{attribute 'enable_dynamic_creation'}
FUNCTION_BLOCK FB_AxisMoveCommand IMPLEMENTS I_Command
VAR
	_Axis : I_Axis;
	_Target : REAL;
	_Description : STRING;
END_VAR

{attribute 'monitoring' := 'call'}
PROPERTY Description : STRING
GET
Description := _Description;
END_GET
END_PROPERTY

METHOD Execute : E_Progress
_Axis.MoveAbsolute(_target);

Execute := E_Progress.Completed;
END_METHOD

//FB_Init is always available implicitly and it is used primarily for initialization.
//The return value is not evaluated. For a specific influence, you can also declare the
//methods explicitly and provide additional code there with the standard initialization
//code. You can evaluate the return value.
METHOD FB_Init: BOOL
VAR_INPUT
    bInitRetains: BOOL; // TRUE: the retain variables are initialized (reset warm / reset cold)
    bInCopyCode: BOOL;  // TRUE: the instance will be copied to the copy code afterward (online change)   
	
	axis : I_Axis;
	target : REAL;
	description : STRING;
END_VAR
_Axis := axis;
_Target := target;
_Description := description;
END_METHOD

METHOD Reset
VAR_INPUT
END_VAR
// nothing to reset here
END_METHOD

END_FUNCTION_BLOCK

(* stored: Version 1.1.0.1
   POU FB_AxisMoveCommand: Id {c26ec26f-d8b8-4f52-ab79-4bfc2dc959d2}, SpecialFunc None
   Property Description: Id {b08bbaba-3238-4666-b36c-e75291820666}
   Get Get: Id {fb223b92-8a32-46ea-874a-048bbfcf52c8}
   Method Execute: Id {3d529086-7b42-47c5-b58f-711b47c0902a}
   Method FB_Init: Id {34bed5db-91fc-4066-a90b-fc405c0eca89}
   Method Reset: Id {c6a07161-05db-43c7-b55a-9ac0a31f9ead} *)
